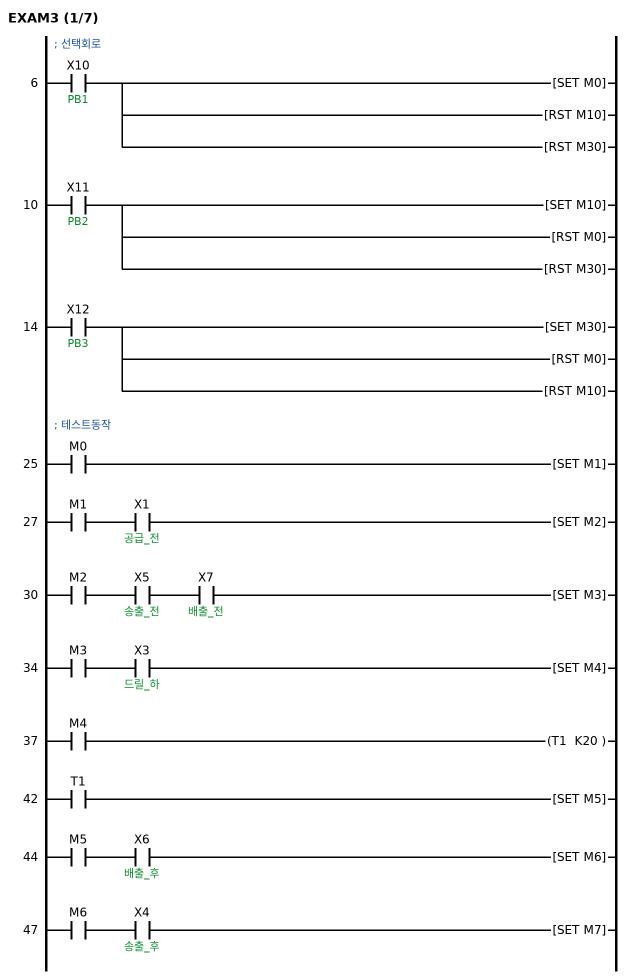
[picture p24: ladder of EXAM3, rungs at steps 6 to 47]
; 선택회로
6     LD      X10  ; PB1
      SET     M0
      RST     M10
      RST     M30
10    LD      X11  ; PB2
      SET     M10
      RST     M0
      RST     M30
14    LD      X12  ; PB3
      SET     M30
      RST     M0
      RST     M10
; 테스트동작
25    LD      M0
      SET     M1
27    LD      M1
      AND     X1  ; 공급_전
      SET     M2
30    LD      M2
      AND     X5  ; 송출_전
      AND     X7  ; 배출_전
      SET     M3
34    LD      M3
      AND     X3  ; 드릴_하
      SET     M4
37    LD      M4
      OUT     T1 K20
42    LD      T1
      SET     M5
44    LD      M5
      AND     X6  ; 배출_후
      SET     M6
47    LD      M6
      AND     X4  ; 송출_후
      SET     M7
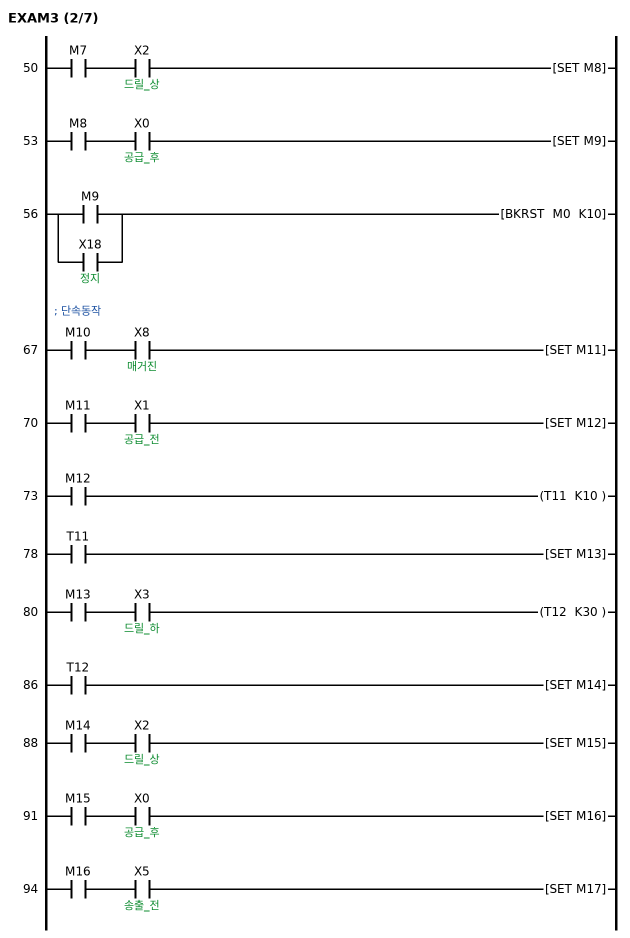
50    LD      M7
      AND     X2  ; 드릴_상
      SET     M8
53    LD      M8
      AND     X0  ; 공급_후
      SET     M9
56    LD      M9
      OR      X18  ; 정지
      BKRST   M0 K10
; 단속동작
67    LD      M10
      AND     X8  ; 매거진
      SET     M11
70    LD      M11
      AND     X1  ; 공급_전
      SET     M12
73    LD      M12
      OUT     T11 K10
78    LD      T11
      SET     M13
80    LD      M13
      AND     X3  ; 드릴_하
      OUT     T12 K30
86    LD      T12
      SET     M14
88    LD      M14
      AND     X2  ; 드릴_상
      SET     M15
91    LD      M15
      AND     X0  ; 공급_후
      SET     M16
94    LD      M16
      AND     X5  ; 송출_전
      SET     M17
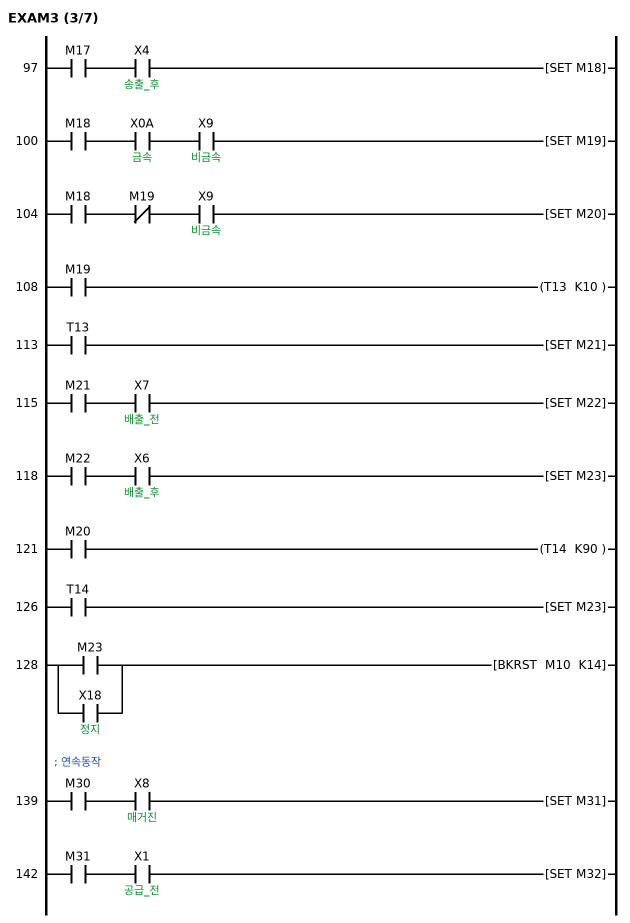
97    LD      M17
      AND     X4  ; 송출_후
      SET     M18
100   LD      M18
      AND     X0A  ; 금속
      AND     X9  ; 비금속
      SET     M19
104   LD      M18
      ANI     M19
      AND     X9  ; 비금속
      SET     M20
108   LD      M19
      OUT     T13 K10
113   LD      T13
      SET     M21
115   LD      M21
      AND     X7  ; 배출_전
      SET     M22
118   LD      M22
      AND     X6  ; 배출_후
      SET     M23
121   LD      M20
      OUT     T14 K90
126   LD      T14
      SET     M23
128   LD      M23
      OR      X18  ; 정지
      BKRST   M10 K14
; 연속동작
139   LD      M30
      AND     X8  ; 매거진
      SET     M31
142   LD      M31
      AND     X1  ; 공급_전
      SET     M32
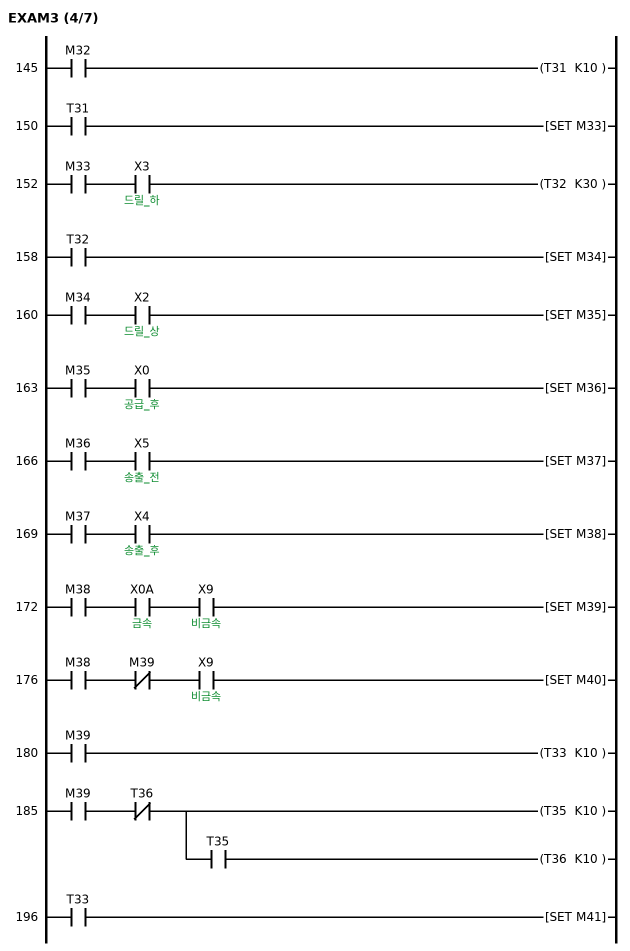
145   LD      M32
      OUT     T31 K10
150   LD      T31
      SET     M33
152   LD      M33
      AND     X3  ; 드릴_하
      OUT     T32 K30
158   LD      T32
      SET     M34
160   LD      M34
      AND     X2  ; 드릴_상
      SET     M35
163   LD      M35
      AND     X0  ; 공급_후
      SET     M36
166   LD      M36
      AND     X5  ; 송출_전
      SET     M37
169   LD      M37
      AND     X4  ; 송출_후
      SET     M38
172   LD      M38
      AND     X0A  ; 금속
      AND     X9  ; 비금속
      SET     M39
176   LD      M38
      ANI     M39
      AND     X9  ; 비금속
      SET     M40
180   LD      M39
      OUT     T33 K10
185   LD      M39
      ANI     T36
      OUT     T35 K10
      AND     T35
      OUT     T36 K10
196   LD      T33
      SET     M41
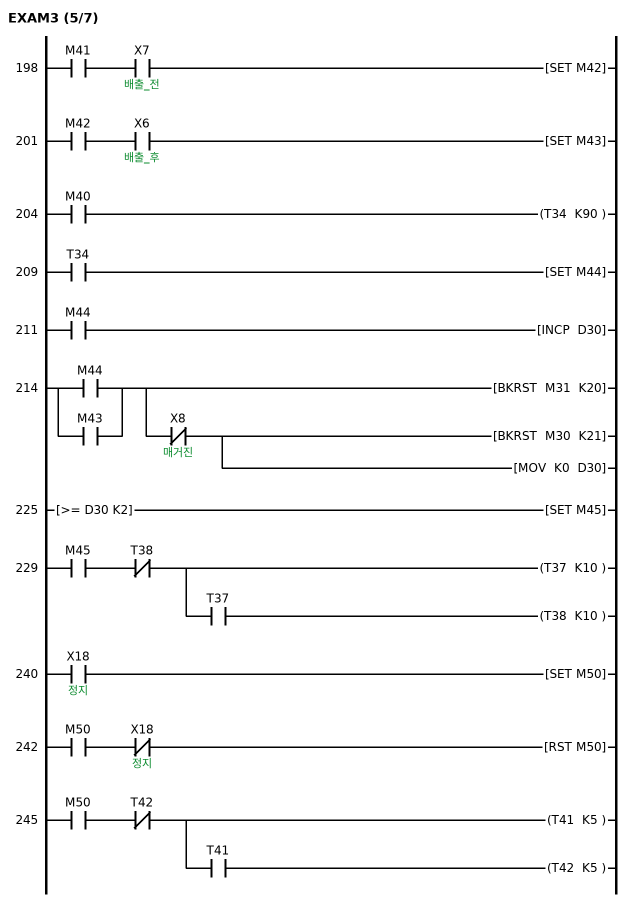
198   LD      M41
      AND     X7  ; 배출_전
      SET     M42
201   LD      M42
      AND     X6  ; 배출_후
      SET     M43
204   LD      M40
      OUT     T34 K90
209   LD      T34
      SET     M44
211   LD      M44
      INCP    D30
214   LD      M44
      OR      M43
      BKRST   M31 K20
      ANI     X8  ; 매거진
      BKRST   M30 K21
      MOV     K0 D30
225   LD>=    D30 K2
      SET     M45
229   LD      M45
      ANI     T38
      OUT     T37 K10
      AND     T37
      OUT     T38 K10
240   LD      X18  ; 정지
      SET     M50
242   LD      M50
      ANI     X18  ; 정지
      RST     M50
245   LD      M50
      ANI     T42
      OUT     T41 K5
      AND     T41
      OUT     T42 K5
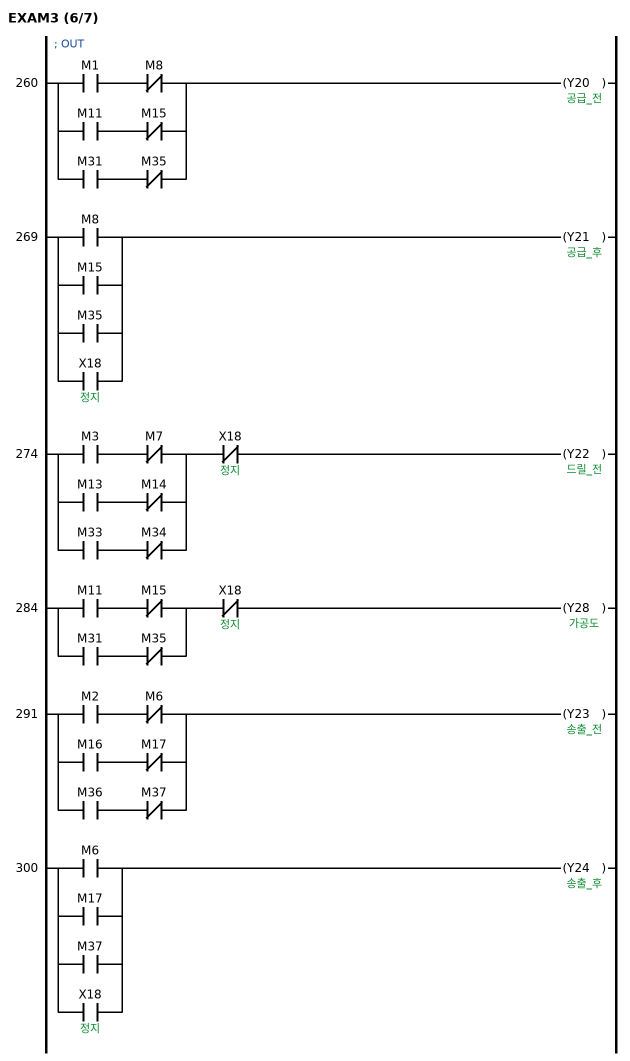
; OUT
260   LD      M1
      ANI     M8
      LD      M11
      ANI     M15
      ORB
      LD      M31
      ANI     M35
      ORB
      OUT     Y20  ; 공급_전
269   LD      M8
      OR      M15
      OR      M35
      OR      X18  ; 정지
      OUT     Y21  ; 공급_후
274   LD      M3
      ANI     M7
      LD      M13
      ANI     M14
      ORB
      LD      M33
      ANI     M34
      ORB
      ANI     X18  ; 정지
      OUT     Y22  ; 드릴_전
284   LD      M11
      ANI     M15
      LD      M31
      ANI     M35
      ORB
      ANI     X18  ; 정지
      OUT     Y28  ; 가공도
291   LD      M2
      ANI     M6
      LD      M16
      ANI     M17
      ORB
      LD      M36
      ANI     M37
      ORB
      OUT     Y23  ; 송출_전
300   LD      M6
      OR      M17
      OR      M37
      OR      X18  ; 정지
      OUT     Y24  ; 송출_후
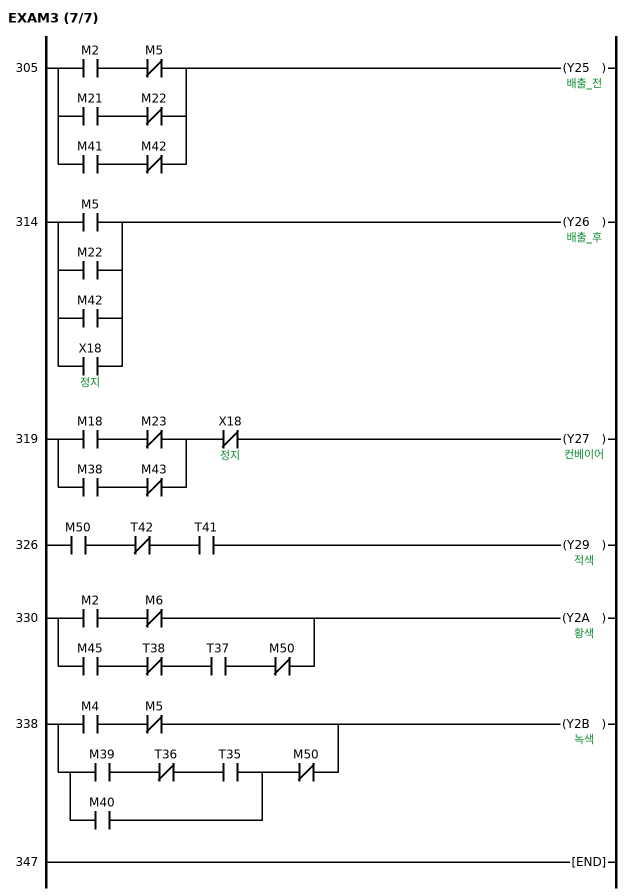
305   LD      M2
      ANI     M5
      LD      M21
      ANI     M22
      ORB
      LD      M41
      ANI     M42
      ORB
      OUT     Y25  ; 배출_전
314   LD      M5
      OR      M22
      OR      M42
      OR      X18  ; 정지
      OUT     Y26  ; 배출_후
319   LD      M18
      ANI     M23
      LD      M38
      ANI     M43
      ORB
      ANI     X18  ; 정지
      OUT     Y27  ; 컨베이어
326   LD      M50
      ANI     T42
      AND     T41
      OUT     Y29  ; 적색
330   LD      M2
      ANI     M6
      LD      M45
      ANI     T38
      AND     T37
      ANI     M50
      ORB
      OUT     Y2A  ; 황색
338   LD      M4
      ANI     M5
      LD      M39
      ANI     T36
      AND     T35
      OR      M40
      ANI     M50
      ORB
      OUT     Y2B  ; 녹색
347   END
END_PROGRAM

PROGRAM EXAM4
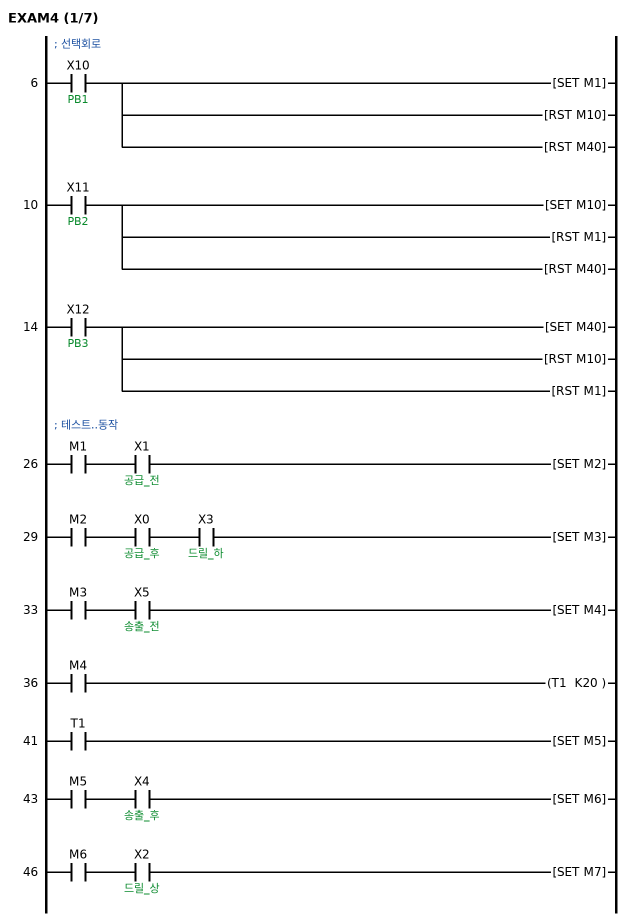
; 선택회로
6     LD      X10  ; PB1
      SET     M1
      RST     M10
      RST     M40
10    LD      X11  ; PB2
      SET     M10
      RST     M1
      RST     M40
14    LD      X12  ; PB3
      SET     M40
      RST     M10
      RST     M1
; 테스트..동작
26    LD      M1
      AND     X1  ; 공급_전
      SET     M2
29    LD      M2
      AND     X0  ; 공급_후
      AND     X3  ; 드릴_하
      SET     M3
33    LD      M3
      AND     X5  ; 송출_전
      SET     M4
36    LD      M4
      OUT     T1 K20
41    LD      T1
      SET     M5
43    LD      M5
      AND     X4  ; 송출_후
      SET     M6
46    LD      M6
      AND     X2  ; 드릴_상
      SET     M7
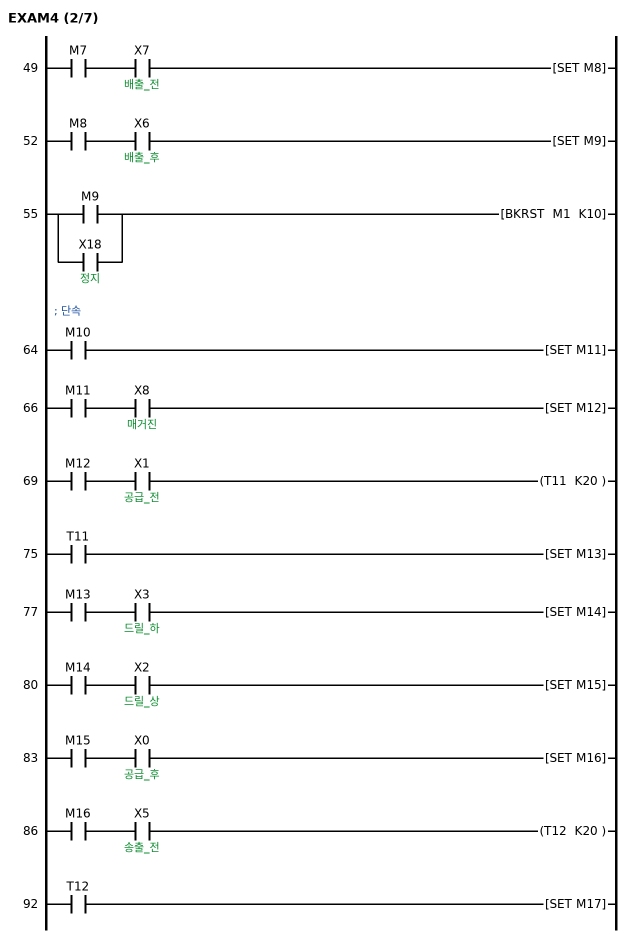
49    LD      M7
      AND     X7  ; 배출_전
      SET     M8
52    LD      M8
      AND     X6  ; 배출_후
      SET     M9
55    LD      M9
      OR      X18  ; 정지
      BKRST   M1 K10
; 단속
64    LD      M10
      SET     M11
66    LD      M11
      AND     X8  ; 매거진
      SET     M12
69    LD      M12
      AND     X1  ; 공급_전
      OUT     T11 K20
75    LD      T11
      SET     M13
77    LD      M13
      AND     X3  ; 드릴_하
      SET     M14
80    LD      M14
      AND     X2  ; 드릴_상
      SET     M15
83    LD      M15
      AND     X0  ; 공급_후
      SET     M16
86    LD      M16
      AND     X5  ; 송출_전
      OUT     T12 K20
92    LD      T12
      SET     M17
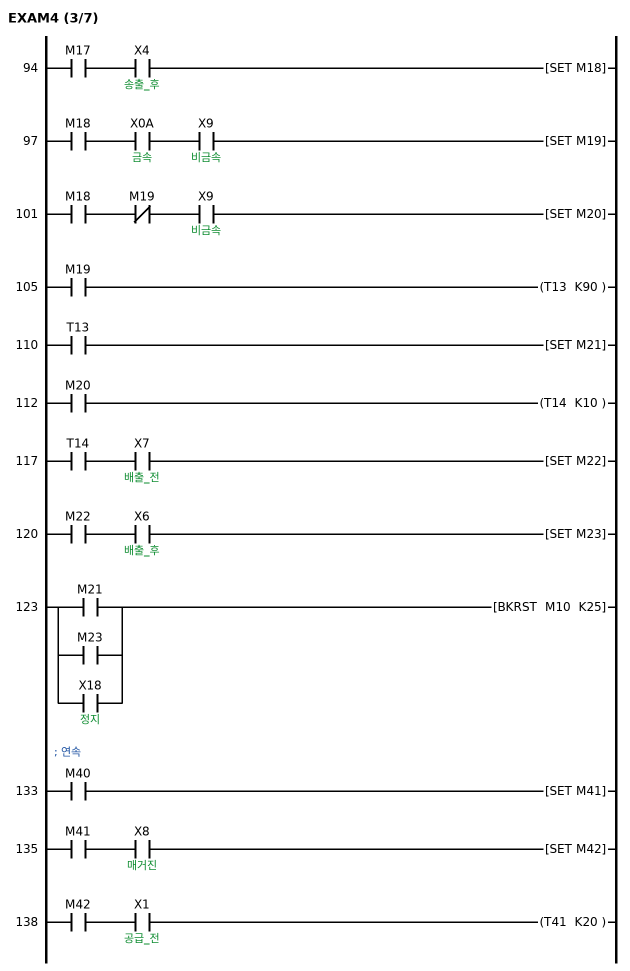
94    LD      M17
      AND     X4  ; 송출_후
      SET     M18
97    LD      M18
      AND     X0A  ; 금속
      AND     X9  ; 비금속
      SET     M19
101   LD      M18
      ANI     M19
      AND     X9  ; 비금속
      SET     M20
105   LD      M19
      OUT     T13 K90
110   LD      T13
      SET     M21
112   LD      M20
      OUT     T14 K10
117   LD      T14
      AND     X7  ; 배출_전
      SET     M22
120   LD      M22
      AND     X6  ; 배출_후
      SET     M23
123   LD      M21
      OR      M23
      OR      X18  ; 정지
      BKRST   M10 K25
; 연속
133   LD      M40
      SET     M41
135   LD      M41
      AND     X8  ; 매거진
      SET     M42
138   LD      M42
      AND     X1  ; 공급_전
      OUT     T41 K20
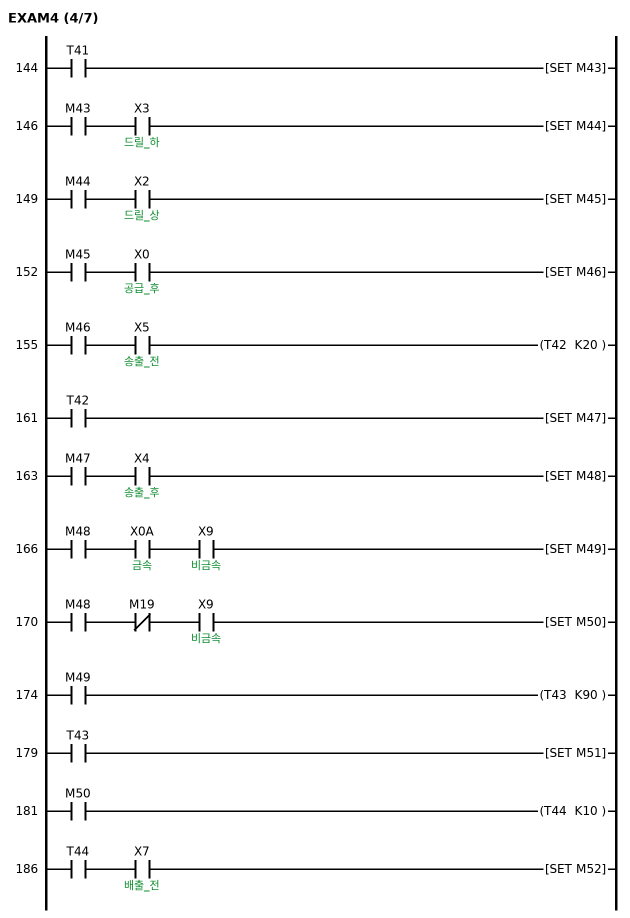
144   LD      T41
      SET     M43
146   LD      M43
      AND     X3  ; 드릴_하
      SET     M44
149   LD      M44
      AND     X2  ; 드릴_상
      SET     M45
152   LD      M45
      AND     X0  ; 공급_후
      SET     M46
155   LD      M46
      AND     X5  ; 송출_전
      OUT     T42 K20
161   LD      T42
      SET     M47
163   LD      M47
      AND     X4  ; 송출_후
      SET     M48
166   LD      M48
      AND     X0A  ; 금속
      AND     X9  ; 비금속
      SET     M49
170   LD      M48
      ANI     M19
      AND     X9  ; 비금속
      SET     M50
174   LD      M49
      OUT     T43 K90
179   LD      T43
      SET     M51
181   LD      M50
      OUT     T44 K10
186   LD      T44
      AND     X7  ; 배출_전
      SET     M52
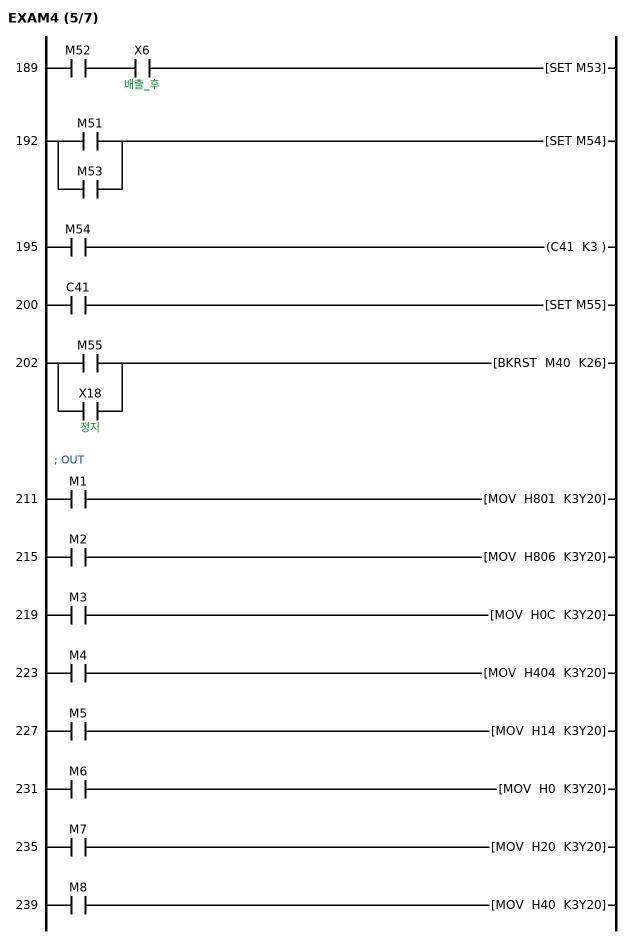
189   LD      M52
      AND     X6  ; 배출_후
      SET     M53
192   LD      M51
      OR      M53
      SET     M54
195   LD      M54
      OUT     C41 K3
200   LD      C41
      SET     M55
202   LD      M55
      OR      X18  ; 정지
      BKRST   M40 K26
; OUT
211   LD      M1
      MOV     H801 K3Y20  ; 공급_전
215   LD      M2
      MOV     H806 K3Y20
219   LD      M3
      MOV     H0C K3Y20
223   LD      M4
      MOV     H404 K3Y20
227   LD      M5
      MOV     H14 K3Y20
231   LD      M6
      MOV     H0 K3Y20
235   LD      M7
      MOV     H20 K3Y20
239   LD      M8
      MOV     H40 K3Y20
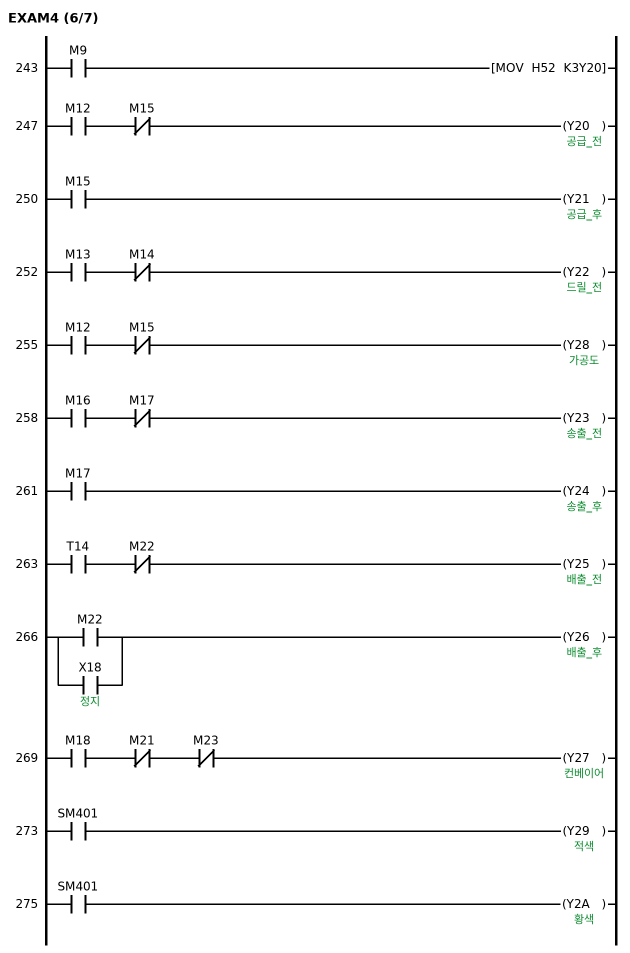
243   LD      M9
      MOV     H52 K3Y20
247   LD      M12
      ANI     M15
      OUT     Y20  ; 공급_전
250   LD      M15
      OUT     Y21  ; 공급_후
252   LD      M13
      ANI     M14
      OUT     Y22  ; 드릴_전
255   LD      M12
      ANI     M15
      OUT     Y28  ; 가공도
258   LD      M16
      ANI     M17
      OUT     Y23  ; 송출_전
261   LD      M17
      OUT     Y24  ; 송출_후
263   LD      T14
      ANI     M22
      OUT     Y25  ; 배출_전
266   LD      M22
      OR      X18  ; 정지
      OUT     Y26  ; 배출_후
269   LD      M18
      ANI     M21
      ANI     M23
      OUT     Y27  ; 컨베이어
273   LD      SM401
      OUT     Y29  ; 적색
275   LD      SM401
      OUT     Y2A  ; 황색
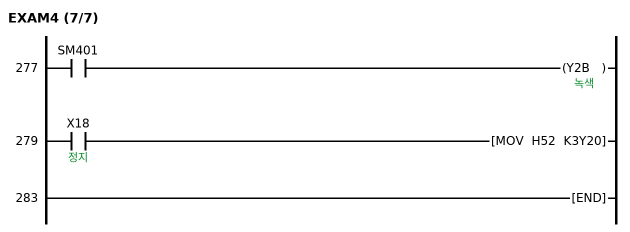
277   LD      SM401
      OUT     Y2B  ; 녹색
279   LD      X18  ; 정지
      MOV     H52 K3Y20
283   END
END_PROGRAM
